LIN {X 0,Y 114.552,Z 541.304,A -85,B 0,C 180,E1 -30776.033,E2 -30776.033} C_VEL
LIN {X 0,Y 119.361,Z 528.742,A -85,B 0,C 180,E1 -30776.414,E2 -30776.414} C_VEL
LIN {X 0,Y 120.719,Z 524.217,A -85,B 0,C 180,E1 -30776.548,E2 -30776.548} C_VEL
LIN {X 0,Y 120.85,Z 522.721,A -85,B 0,C 180,E1 -30780,E2 -30780} C_VEL
LIN {X 0,Y 120.613,Z 524.232,A -85,B 0,C 180,E1 -30783.998,E2 -30783.998} C_VEL
LIN {X 0,Y 116.354,Z 536.715,A -85,B 0,C 180,E1 -30784.617,E2 -30784.617} C_VEL
LIN {X 0,Y 111.148,Z 547.997,A -85,B 0,C 180,E1 -30785.215,E2 -30785.215} C_VEL
LIN {X 0,Y 104.246,Z 559.59,A -85,B 0,C 180,E1 -30786.074,E2 -30786.074} C_VEL
LIN {X 0,Y 96.495,Z 570.01,A -85,B 0,C 180,E1 -30787.104,E2 -30787.104} C_VEL
LIN {X 0,Y 88.788,Z 578.521,A -85,B 0,C 180,E1 -30788.344,E2 -30788.344} C_VEL
LIN {X 0,Y 79.701,Z 586.854,A -85,B 0,C 180,E1 -30790.158,E2 -30790.158} C_VEL
LIN {X 0,Y 70.196,Z 594.007,A -85,B 0,C 180,E1 -30792.54,E2 -30792.54} C_VEL
LIN {X 0,Y 61.864,Z 599.238,A -85,B 0,C 180,E1 -30795.07,E2 -30795.07} C_VEL
LIN {X 0,Y 52.035,Z 604.309,A -85,B 0,C 180,E1 -30799.017,E2 -30799.017} C_VEL
LIN {X 0,Y 42.642,Z 608.234,A -85,B 0,C 180,E1 -30804.979,E2 -30804.979} C_VEL
LIN {X 0,Y 33.89,Z 611.128,A -85,B 0,C 180,E1 -30813.955,E2 -30813.955} C_VEL
LIN {X 0,Y 24.332,Z 613.487,A -85,B 0,C 180,E1 -30834.714,E2 -30834.714} C_VEL
LIN {X 0,Y 23.888,Z 613.559,A -85,B 0,C 180,E1 -30836.425,E2 -30836.425} C_VEL
LIN {X 0,Y 21.822,Z 613.948,A -85,B 0,C 180,E1 -30844.824,E2 -30844.824} C_VEL
LIN {X 0,Y 18.854,Z 614.323,A -85,B 0,C 180,E1 -30859.358,E2 -30859.358} C_VEL
LIN {X 0,Y 17.109,Z 614.152,A -85,B 0,C 180,E1 -30904.817,E2 -30904.817} C_VEL
LIN {X 0,Y 20.118,Z 613.62,A -85,B 0,C 180,E1 -30920.718,E2 -30920.718} C_VEL
LIN {X 0,Y 21.559,Z 613.314,A -85,B 0,C 180,E1 -30924.436,E2 -30924.436} C_VEL
LIN {X 0,Y 30.485,Z 611.473,A -85,B 0,C 180,E1 -30937.241,E2 -30937.241} C_VEL
LIN {X 0,Y 40.154,Z 608.608,A -85,B 0,C 180,E1 -30944.285,E2 -30944.285} C_VEL
LIN {X 0,Y 50.159,Z 604.722,A -85,B 0,C 180,E1 -30948.747,E2 -30948.747} C_VEL
LIN {X 0,Y 60.395,Z 599.694,A -85,B 0,C 180,E1 -30951.535,E2 -30951.535} C_VEL
LIN {X 0,Y 70.71,Z 593.361,A -85,B 0,C 180,E1 -30953.664,E2 -30953.664} C_VEL
LIN {X 0,Y 81.079,Z 585.447,A -85,B 0,C 180,E1 -30955.417,E2 -30955.417} C_VEL
LIN {X 0,Y 89.769,Z 577.37,A -85,B 0,C 180,E1 -30956.54,E2 -30956.54} C_VEL
LIN {X 0,Y 98.488,Z 567.507,A -85,B 0,C 180,E1 -30957.438,E2 -30957.438} C_VEL
LIN {X 0,Y 106.352,Z 556.384,A -85,B 0,C 180,E1 -30958.144,E2 -30958.144} C_VEL
LIN {X 0,Y 113.159,Z 544.109,A -85,B 0,C 180,E1 -30958.659,E2 -30958.659} C_VEL
LIN {X 0,Y 118.062,Z 532.557,A -85,B 0,C 180,E1 -30959.12,E2 -30959.12} C_VEL
LIN {X 0,Y 118.643,Z 530.876,A -85,B 0,C 180,E1 -30959.165,E2 -30959.165} C_VEL
LIN {X 0,Y 118.936,Z 530.008,A -85,B 0,C 180,E1 -30959.553,E2 -30959.553} C_VEL
LIN {X 0,Y 118.946,Z 530.003,A -85,B 0,C 180,E1 -30960,E2 -30960} C_VEL
LIN {X 0,Y 118.666,Z 530.854,A -85,B 0,C 180,E1 -30960.248,E2 -30960.248} C_VEL
LIN {X 0,Y 113.852,Z 542.767,A -85,B 0,C 180,E1 -30960.464,E2 -30960.464} C_VEL
LIN {X 0,Y 108.062,Z 553.712,A -85,B 0,C 180,E1 -30960.734,E2 -30960.734} C_VEL
LIN {X 0,Y 100.168,Z 565.461,A -85,B 0,C 180,E1 -30961.181,E2 -30961.181} C_VEL
LIN {X 0,Y 91.407,Z 575.893,A -85,B 0,C 180,E1 -30961.799,E2 -30961.799} C_VEL
LIN {X 0,Y 82.661,Z 584.343,A -85,B 0,C 180,E1 -30962.59,E2 -30962.59} C_VEL
LIN {X 0,Y 72.196,Z 592.602,A -85,B 0,C 180,E1 -30963.828,E2 -30963.828} C_VEL
LIN {X 0,Y 61.791,Z 599.268,A -85,B 0,C 180,E1 -30965.62,E2 -30965.62} C_VEL
LIN {X 0,Y 49.784,Z 605.375,A -85,B 0,C 180,E1 -30968.826,E2 -30968.826} C_VEL
LIN {X 0,Y 39.663,Z 609.35,A -85,B 0,C 180,E1 -30972.959,E2 -30972.959} C_VEL
LIN {X 0,Y 29.849,Z 612.292,A -85,B 0,C 180,E1 -30979.648,E2 -30979.648} C_VEL
LIN {X 0,Y 18.289,Z 614.711,A -85,B 0,C 180,E1 -30999.777,E2 -30999.777} C_VEL
LIN {X 0,Y 14.253,Z 615.334,A -85,B 0,C 180,E1 -31020.458,E2 -31020.458} C_VEL
LIN {X 0,Y 12.975,Z 615.559,A -85,B 0,C 180,E1 -31050,E2 -31050} C_VEL
LIN {X 0,Y 14.253,Z 615.312,A -85,B 0,C 180,E1 -31079.543,E2 -31079.543} C_VEL
LIN {X 0,Y 18.288,Z 614.676,A -85,B 0,C 180,E1 -31100.226,E2 -31100.226} C_VEL
LIN {X 0,Y 29.849,Z 612.221,A -85,B 0,C 180,E1 -31120.356,E2 -31120.356} C_VEL
LIN {X 0,Y 39.663,Z 609.249,A -85,B 0,C 180,E1 -31127.04,E2 -31127.04} C_VEL
LIN {X 0,Y 49.794,Z 605.241,A -85,B 0,C 180,E1 -31131.101,E2 -31131.101} C_VEL
LIN {X 0,Y 61.799,Z 599.081,A -85,B 0,C 180,E1 -31134.301,E2 -31134.301} C_VEL
LIN {X 0,Y 72.198,Z 592.37,A -85,B 0,C 180,E1 -31136.15,E2 -31136.15} C_VEL
LIN {X 0,Y 82.663,Z 584.061,A -85,B 0,C 180,E1 -31137.39,E2 -31137.39} C_VEL
LIN {X 0,Y 91.407,Z 575.535,A -85,B 0,C 180,E1 -31138.202,E2 -31138.202} C_VEL
LIN {X 0,Y 100.168,Z 565.01,A -85,B 0,C 180,E1 -31138.825,E2 -31138.825} C_VEL
LIN {X 0,Y 108.061,Z 553.16,A -85,B 0,C 180,E1 -31139.286,E2 -31139.286} C_VEL
LIN {X 0,Y 114.46,Z 540.623,A -85,B 0,C 180,E1 -31139.6,E2 -31139.6} C_VEL
LIN {X 0,Y 118.39,Z 530.653,A -85,B 0,C 180,E1 -31139.788,E2 -31139.788} C_VEL
LIN {X 0,Y 118.727,Z 529.637,A -85,B 0,C 180,E1 -31140,E2 -31140} C_VEL
LIN {X 0,Y 118.707,Z 529.669,A -85,B 0,C 180,E1 -31140.493,E2 -31140.493} C_VEL
LIN {X 0,Y 118.132,Z 531.369,A -85,B 0,C 180,E1 -31140.918,E2 -31140.918} C_VEL
LIN {X 0,Y 113.089,Z 543.563,A -85,B 0,C 180,E1 -31141.356,E2 -31141.356} C_VEL
LIN {X 0,Y 106.359,Z 555.825,A -85,B 0,C 180,E1 -31141.967,E2 -31141.967} C_VEL
LIN {X 0,Y 98.495,Z 567.082,A -85,B 0,C 180,E1 -31142.652,E2 -31142.652} C_VEL
LIN {X 0,Y 89.777,Z 577.018,A -85,B 0,C 180,E1 -31143.544,E2 -31143.544} C_VEL
LIN {X 0,Y 81.092,Z 585.153,A -85,B 0,C 180,E1 -31144.722,E2 -31144.722} C_VEL
LIN {X 0,Y 70.722,Z 593.117,A -85,B 0,C 180,E1 -31146.423,E2 -31146.423} C_VEL
LIN {X 0,Y 60.41,Z 599.507,A -85,B 0,C 180,E1 -31148.56,E2 -31148.56} C_VEL
LIN {X 0,Y 50.173,Z 604.577,A -85,B 0,C 180,E1 -31151.33,E2 -31151.33} C_VEL
LIN {X 0,Y 40.163,Z 608.502,A -85,B 0,C 180,E1 -31155.761,E2 -31155.761} C_VEL
LIN {X 0,Y 30.493,Z 611.396,A -85,B 0,C 180,E1 -31162.796,E2 -31162.796} C_VEL
LIN {X 0,Y 24.422,Z 612.775,A -85,B 0,C 180,E1 -31170.311,E2 -31170.311} C_VEL
LIN {X 0,Y 14.877,Z 614.352,A -85,B 0,C 180,E1 -31201.809,E2 -31201.809} C_VEL
LIN {X 0,Y 13.306,Z 614.57,A -85,B 0,C 180,E1 -31230,E2 -31230} C_VEL
LIN {X 0,Y 14.877,Z 614.375,A -85,B 0,C 180,E1 -31258.191,E2 -31258.191} C_VEL
LIN {X 0,Y 21.559,Z 613.314,A -85,B 0,C 180,E1 -31284.436,E2 -31284.436} C_VEL
LIN {X 0,Y 25.965,Z 612.482,A -85,B 0,C 180,E1 -31293.755,E2 -31293.755} C_VEL
LIN {X 0,Y 33.295,Z 610.587,A -85,B 0,C 180,E1 -31306.327,E2 -31306.327} C_VEL
LIN {X 0,Y 41.423,Z 608.016,A -85,B 0,C 180,E1 -31314.236,E2 -31314.236} C_VEL
LIN {X 0,Y 46.748,Z 606.007,A -85,B 0,C 180,E1 -31316.379,E2 -31316.379} C_VEL
LIN {X 0,Y 59.764,Z 599.959,A -85,B 0,C 180,E1 -31318.275,E2 -31318.275} C_VEL
LIN {X 0,Y 63.264,Z 597.985,A -85,B 0,C 180,E1 -31318.808,E2 -31318.808} C_VEL
LIN {X 0,Y 52.623,Z 603.553,A -85,B 0,C 180,E1 -31320,E2 -31320} C_VEL
LIN {X 0,Y 42.188,Z 607.857,A -85,B 0,C 180,E1 -31321.819,E2 -31321.819} C_VEL
LIN {X 0,Y 35.207,Z 610.161,A -85,B 0,C 180,E1 -31323.556,E2 -31323.556} C_VEL
LIN {X 0,Y 28.262,Z 612.025,A -85,B 0,C 180,E1 -31325.923,E2 -31325.923} C_VEL
LIN {X 0,Y 14.78,Z 614.443,A -85,B 0,C 180,E1 -31338.01,E2 -31338.01} C_VEL
LIN {X 0,Y 8.794,Z 615.067,A -85,B 0,C 180,E1 -31356.954,E2 -31356.954} C_VEL
LIN {X 0,Y 5.879,Z 615.292,A -85,B 0,C 180,E1 -31410,E2 -31410} C_VEL
LIN {X 0,Y 8.794,Z 615.044,A -85,B 0,C 180,E1 -31463.049,E2 -31463.049} C_VEL
LIN {X 0,Y 14.779,Z 614.407,A -85,B 0,C 180,E1 -31481.995,E2 -31481.995} C_VEL
LIN {X 0,Y 28.262,Z 611.952,A -85,B 0,C 180,E1 -31494.081,E2 -31494.081} C_VEL
LIN {X 0,Y 38.692,Z 608.979,A -85,B 0,C 180,E1 -31497.418,E2 -31497.418} C_VEL
LIN {X 0,Y 49.198,Z 604.97,A -85,B 0,C 180,E1 -31499.37,E2 -31499.37} C_VEL
LIN {X 0,Y 61.502,Z 598.81,A -85,B 0,C 180,E1 -31500.951,E2 -31500.951} C_VEL
LIN {X 0,Y 63.263,Z 597.794,A -85,B 0,C 180,E1 -31501.14,E2 -31501.14} C_VEL
LIN {X 0,Y 63.271,Z 597.781,A -85,B 0,C 180,E1 -31501.449,E2 -31501.449} C_VEL
LIN {X 0,Y 51.537,Z 603.827,A -85,B 0,C 180,E1 -31502.88,E2 -31502.88} C_VEL
LIN {X 0,Y 38.841,Z 608.77,A -85,B 0,C 180,E1 -31505.635,E2 -31505.635} C_VEL
LIN {X 0,Y 28.503,Z 611.664,A -85,B 0,C 180,E1 -31509.511,E2 -31509.511} C_VEL
LIN {X 0,Y 21.724,Z 613.042,A -85,B 0,C 180,E1 -31513.948,E2 -31513.948} C_VEL
LIN {X 0,Y 9.247,Z 614.619,A -85,B 0,C 180,E1 -31540.536,E2 -31540.536} C_VEL
LIN {X 0,Y 6.211,Z 614.837,A -85,B 0,C 180,E1 -31590,E2 -31590} C_VEL
LIN {X 0,Y 9.247,Z 614.642,A -85,B 0,C 180,E1 -31639.465,E2 -31639.465} C_VEL
LIN {X 0,Y 21.722,Z 613.094,A -85,B 0,C 180,E1 -31666.07,E2 -31666.07} C_VEL
LIN {X 0,Y 28.5,Z 611.739,A -85,B 0,C 180,E1 -31670.529,E2 -31670.529} C_VEL
LIN {X 0,Y 38.837,Z 608.874,A -85,B 0,C 180,E1 -31674.417,E2 -31674.417} C_VEL
LIN {X 0,Y 46.748,Z 606.007,A -85,B 0,C 180,E1 -31676.379,E2 -31676.379} C_VEL
LIN {X 0,Y 46.748,Z 606.007,A -85,B 0,C 180,E1 -31676.379,E2 -31676.379}

QRS_NEXT_CUT()

QRS_NEXT()
QRS_HOME()

END
